TYPE MQTTSettings :
STRUCT
	//Broker info
	brokerIP : STRING := '78.27.125.143';
    brokerPort : UINT := 8885;
	brokerUsername : STRING := 'scanrobot';
	brokerPassword : STRING := 'kissa';
	
	//Client info
    clientId : STRING := 'plc';
	topicPub : STRING := 'beckhoff';
	topicSub : STRING := 'beckhoff';
	qos : TcIotMqttQos := TcIotMqttQos.AtMostOnceDelivery;	
	
	//TLS info
	caCertificateAbsolutePath : STRING := 'C:\Users\mikko\Desktop\folders\projects\scan_robot\twincat\certs\ca.crt';
	clientCertificateAbsolutePath : STRING := 'C:\Users\mikko\Desktop\folders\projects\scan_robot\twincat\certs\client.crt';
	clientKeyAbsolutePath : STRING := 'C:\Users\mikko\Desktop\folders\projects\scan_robot\twincat\certs\client.key';
END_STRUCT
END_TYPE

(* stored: Version 1.1.0.1, ProductVersion 3.1.4024.11
   DUT MQTTSettings: Id {c150fbe4-de94-4c4b-bc27-8cb0c2fadd85} *)
